// TIA Portal V20 export
TYPE "typeOpLampStatus"
// stored: Access Published, IsFailsafeCompliant true, Namespace Safety
   STRUCT
      InitializeEnable : Bool;
      HomeLampStatus : Bool;
      LampStatus2 : Bool;
      LampStatus3 : Bool;
      LampStatus4 : Bool;
      LampStatus5 : Bool;
      LampStatus6 : Bool;
   END_STRUCT;
END_TYPE
